(* IEC 61131-3 sources: lsinatopo/src, 1 file *)

(* ---- myClass.st ---- *)
NAMESPACE Simatic.Ax.lsinatopo

    {axcode:docs-v0:@simatic-ax/lsinatopo:MyClass.md}
    CLASS MyClass

        VAR PUBLIC
        END_VAR

        VAR
        END_VAR

        /// Inline Comment for MyMethod. It will be shown, when you hover over the method
        /// This method has no parameters and no return value
        METHOD PUBLIC MyMethod
            ;
        END_METHOD

    END_CLASS

END_NAMESPACE
